SUBAPPLICATION SIFB100 (* Subapplication Type *)
  (* Standard: 61499-2 *)
  (* Version 1.0, 2025-05-03, cochicde *)
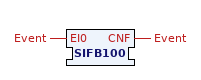
  EVENT_INPUT
    EI0;
  END_EVENT
  EVENT_OUTPUT
    CNF;
  END_EVENT
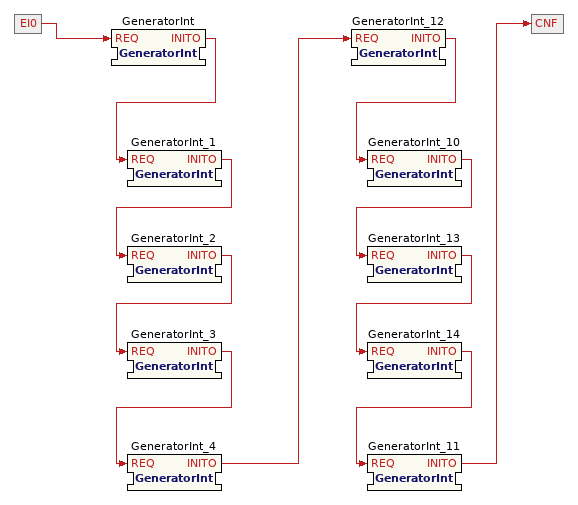
  FBS
    GeneratorInt_2 : performance::GeneratorInt;
    GeneratorInt_1 : performance::GeneratorInt;
    GeneratorInt_3 : performance::GeneratorInt;
    GeneratorInt : performance::GeneratorInt;
    GeneratorInt_4 : performance::GeneratorInt;
    GeneratorInt_10 : performance::GeneratorInt;
    GeneratorInt_11 : performance::GeneratorInt;
    GeneratorInt_12 : performance::GeneratorInt;
    GeneratorInt_13 : performance::GeneratorInt;
    GeneratorInt_14 : performance::GeneratorInt;
  END_FBS
  EVENT_CONNECTIONS
    EI0 TO GeneratorInt.REQ;
    GeneratorInt_1.INITO TO GeneratorInt_2.REQ;
    GeneratorInt_3.INITO TO GeneratorInt_4.REQ;
    GeneratorInt_2.INITO TO GeneratorInt_3.REQ;
    GeneratorInt.INITO TO GeneratorInt_1.REQ;
    GeneratorInt_13.INITO TO GeneratorInt_14.REQ;
    GeneratorInt_10.INITO TO GeneratorInt_13.REQ;
    GeneratorInt_14.INITO TO GeneratorInt_11.REQ;
    GeneratorInt_12.INITO TO GeneratorInt_10.REQ;
    GeneratorInt_4.INITO TO GeneratorInt_12.REQ;
    GeneratorInt_11.INITO TO CNF;
  END_CONNECTIONS
END_SUBAPPLICATION
